PROGRAM MAIN
VAR
	Estacion: FB_Estacion;
END_VAR

Estacion();

END_PROGRAM

(* stored: Version 1.1.0.1, ProductVersion 3.1.4024.12
   POU MAIN: Id {ac507533-9318-47ac-91b7-94a836fda366}, SpecialFunc None *)
